// Implicitly generated code : DO NOT EDIT
FUNCTION CheckBounds : DINT
VAR_INPUT
	index, lower, upper: DINT;
END_VAR
VAR_STAT
	counter:int;
END_VAR

// Implicitly generated code : Only an Implementation suggestion
{noflow}
IF  index < lower THEN
	CheckBounds := lower;
	counter:=counter+1;
ELSIF  index > upper THEN
	CheckBounds := upper;
	counter:=counter+1;
ELSE  
	CheckBounds := index;
END_IF
{flow}

END_FUNCTION

(* stored: Version 1.1.0.1, ProductVersion 3.1.4024.10
   POU CheckBounds: Id {4f8d0503-95c8-4a6d-897f-2267b0b6a76b}, SpecialFunc CheckBounds *)
